// Miscellaneous.
FUNCTION_BLOCK FB_Misc EXTENDS FB_BA_View
VAR	
	// Intention:		Take care of UTF-8 encoding manually.
	//					> [Hint] Disable the integrated encoding mechanism (See "BA_Param.bUtf8AutoConvert")!
	SpecialUtf8			: FB_BA_AV_Op := (
							iParent					:= THIS^,
							sDescription			:= wsLiteral_TO_UTF8("{äöüßéèêµ€° Ἀθῆναι İstanbul Київ}"),
							eUnit					:= E_BA_Unit.eOther_Percent,
							fValueRm				:= 5
						);
END_VAR

SUPER^();

SpecialUtf8();

END_FUNCTION_BLOCK

(* stored: Version 1.1.0.1, ProductVersion 3.1.4024.11
   POU FB_Misc: Id {3ab59abd-7907-417e-9172-68b9f3ae54be}, SpecialFunc None *)
